{attribute 'no_explicit_call' := 'Body contains no logic, calling methods only allowed.'}
{attribute 'hide_all_locals'}

// A class containing possible gas types for Bronkhorst devices stored as a string.
PROGRAM GasTypes
VAR
END_VAR

{attribute 'monitoring':='call}
PROPERTY Air : STRING
GET
Air := 'AiR';
END_GET
END_PROPERTY

{attribute 'monitoring':='variable'}
PROPERTY BBr3 : STRING
GET
BBr3 := 'BBr3';
END_GET
END_PROPERTY

{attribute 'monitoring':='variable'}
PROPERTY BCl3 : STRING
GET
BCl3 := 'BCl3';
END_GET
END_PROPERTY

{attribute 'monitoring':='variable'}
PROPERTY C2F6 : STRING
GET
C2F6 := 'C2F6';
END_GET
END_PROPERTY

{attribute 'monitoring':='variable'}
PROPERTY Cl2 : STRING
GET
Cl2 := 'Cl2';
END_GET
END_PROPERTY

{attribute 'monitoring':='variable'}
PROPERTY H2 : STRING
GET
H2 := 'H2';
END_GET
END_PROPERTY

{attribute 'monitoring':='variable'}
PROPERTY He : STRING
GET
He := 'He';
END_GET
END_PROPERTY

{attribute 'monitoring':='variable'}
PROPERTY N2 : STRING
GET
N2 := 'N2';
END_GET
END_PROPERTY

{attribute 'monitoring':='variable'}
PROPERTY O2 : STRING
GET
O2 := 'O2';
END_GET
END_PROPERTY

{attribute 'monitoring':='variable'}
PROPERTY SF6 : STRING
GET
SF6 := 'SF6';
END_GET
END_PROPERTY

{attribute 'monitoring':='variable'}
PROPERTY SiF4 : STRING
GET
SiF4 := 'SiF4';
END_GET
END_PROPERTY

END_PROGRAM

(* stored: Version 1.1.0.1
   POU GasTypes: Id {29a0b4bc-11ec-0b5c-1f68-73f742326369}, SpecialFunc None
   Property Air: Id {0f26b01b-994b-0bc1-2d5a-3515f6e948fe}
   Get Get: Id {4da449fa-493a-03bb-2aa4-59155281b4c6}
   Property BBr3: Id {328611a6-b1b7-0214-0e93-e90a6fdd79ea}
   Get Get: Id {1eee6602-765c-0afb-073e-c7c38414ff74}
   Property BCl3: Id {5d338191-fefc-0be6-0c03-23da561f9d85}
   Get Get: Id {b8fce984-c912-0f9f-1de5-0b1762e5087c}
   Property C2F6: Id {f2ef586f-0e5b-0659-29bb-1a25e927e282}
   Get Get: Id {1a0dc294-c17d-09c8-1a8c-e71fa91d9654}
   Property Cl2: Id {445322bc-5b50-0dfc-0d6c-0de2399852f8}
   Get Get: Id {4bd06be8-29c9-0cac-2b53-bdebe893828b}
   Property H2: Id {c8691a1c-8cc5-0f8d-0df4-a2109971f2e9}
   Get Get: Id {bd00b772-2e9d-0c9a-01f7-45b5753a6c00}
   Property He: Id {8f74035e-bac9-001e-3659-f3c7c9f08775}
   Get Get: Id {7a09f7e9-86b5-0678-1d6c-abae167f6df1}
   Property N2: Id {edad31b3-91ea-09c3-1975-a51b0bf7e2b2}
   Get Get: Id {a8e1d404-9646-0d6b-3281-df4fba58c4ac}
   Property O2: Id {4bcb2d58-a78a-0681-1b48-64ac277d1283}
   Get Get: Id {a2fe2990-e8ca-086f-24cc-66245106486e}
   Property SF6: Id {1bcafec4-6590-0cd1-0934-41699cf18ec5}
   Get Get: Id {b8fd5d71-6f1a-061f-1824-a4240c6b5ca6}
   Property SiF4: Id {faa5f6df-73ba-0629-2622-92d1b18aaba3}
   Get Get: Id {de523e24-f157-0efb-29cb-1bebed9b6d71} *)
